FUNCTION FC_HMIRead : STRING
VAR_INPUT
	linput : LREAL;
	inumber : INT;
END_VAR
VAR
END_VAR

FC_HMIRead := LREAL_TO_FMTSTR(linput,inumber,TRUE);

END_FUNCTION

(* stored: Version 1.1.0.1, ProductVersion 3.1.4024.13
   POU FC_HMIRead: Id {01703944-4b8a-4371-b296-8120e318af3c}, SpecialFunc None *)
